FUNCTION_BLOCK StationCtrl2 (* Template for a simple Basic Function Block Type *)
  (* Standard: 61499-2 *)
  (* Version 1.0, 2020-08-10, AK115394 *)
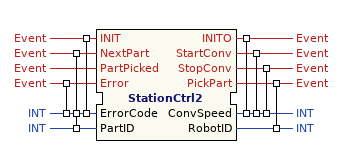
  EVENT_INPUT
    INIT WITH ErrorCode; (* Initialization Request *)
    NextPart WITH PartID, ErrorCode; (* Next part is ready *)
    PartPicked;
    Error WITH ErrorCode; (* Error in system occurred *)
  END_EVENT
  EVENT_OUTPUT
    INITO WITH ConvSpeed; (* Initialization Confirm *)
    StartConv WITH ConvSpeed; (* Execution Confirmation *)
    StopConv WITH ConvSpeed;
    PickPart WITH RobotID;
  END_EVENT
  VAR_INPUT
    ErrorCode : INT; (* Origin and type of error *)
    PartID : INT;
  END_VAR
  VAR_OUTPUT
    ConvSpeed : INT := 100; (* Output event qualifier *)
    RobotID : INT;
  END_VAR
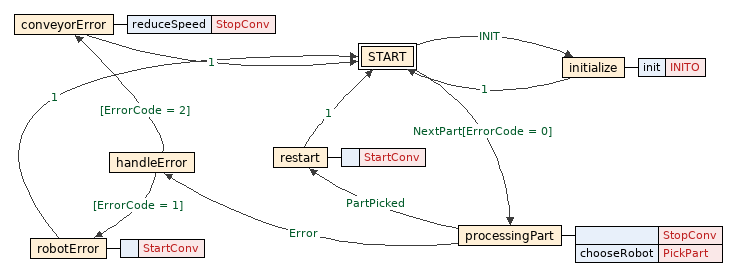
  EC_STATES
    START; (* Initial State *)
    initialize : init -> INITO;
    processingPart : -> StopConv, chooseRobot -> PickPart;
    handleError;
    conveyorError : reduceSpeed -> StopConv;
    robotError : -> StartConv;
    restart : -> StartConv;
  END_STATES
  EC_TRANSITIONS
    START TO initialize := INIT;
    initialize TO START := 1;
    START TO processingPart := NextPart[ErrorCode = 0];
    processingPart TO restart := PartPicked;
    processingPart TO handleError := Error;
    handleError TO robotError := [ErrorCode = 1];
    handleError TO conveyorError := [ErrorCode = 2];
    conveyorError TO START := 1;
    robotError TO START := 1;
    restart TO START := 1;
  END_TRANSITIONS
  ALGORITHM init IN ST:
RobotID := 0;
  END_ALGORITHM
  ALGORITHM setSpeed IN ST:
ConvSpeed := 100;
  END_ALGORITHM
  ALGORITHM chooseRobot IN ST:
RobotID := 50;
  END_ALGORITHM
  ALGORITHM reduceSpeed IN ST:
ConvSpeed := 50;
  END_ALGORITHM
  SERVICE FB Network/BFB Internal
    SEQUENCE initialize {SET_ATTRIBUTE(StartState, START)}
      FB Network.INIT() -> BFB Internal.init() -> FB Network.INITO();
    END_SEQUENCE
    SEQUENCE normal_operation {SET_ATTRIBUTE(StartState, START)}
      FB Network.NextPart(ErrorCode:=0) -> BFB Internal.chooseRobot() -> FB Network.StopConv() -> FB Network.PickPart(ConvSpeed:=INT#100);
      FB Network.PartPicked() -> FB Network.StartConv();
    END_SEQUENCE
    SEQUENCE conveyor_error {SET_ATTRIBUTE(StartState, processingPart)}
      FB Network.Error(ErrorCode:=2) -> BFB Internal.reduceSpeed() -> FB Network.StopConv(ConvSpeed:=50);
    END_SEQUENCE
  END_SERVICE
END_FUNCTION_BLOCK
